{attribute 'GeneratedUsingTerminal: EL4732-0001-0000'}
{attribute addProperty BoxType "EL4732-0001-0000"}
{attribute addProperty Id "Value1AT %Q*INT2Value2AT %Q*INT2"}
{attribute addProperty CRC "3024272229"}
{attribute addProperty Size "4"}
TYPE Sample_B442BB65 EXTENDS OutputBase_10CEE7DE :
STRUCT
	{attribute addProperty Name "Value1"}
	Value1 AT %Q* : INT;
	{attribute addProperty Name "Value2"}
	Value2 AT %Q* : INT;
END_STRUCT
END_TYPE

(* stored: Version 1.2.0.0, ProductVersion 3.1.4024.11
   DUT Sample_B442BB65: Id {f4f3ed14-7257-4708-a8d8-9032013cb4b0} *)
